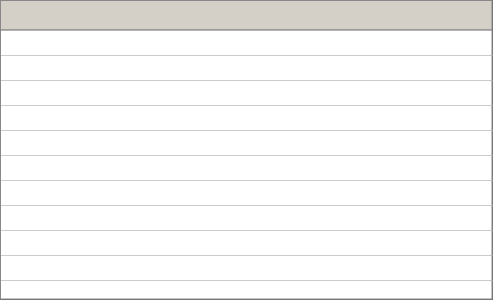
VISUALIZATION _VISU_SRS  // 493x300
VAR_IN_OUT
	mInst : FB_SRS;
END_VAR
    Table (0,0 493x300), data array: mInst.sSrsList
        p3854506369: mInst.sSrsList[INDEX].bImplemented
        p1892666644: mInst.sSrsList[INDEX].sKey
        p338671338: mInst.sSrsList[INDEX].sDescription
        p2170511999: mInst.sSrsList[INDEX].sLink
        p2232123230: Impl.
END_VISUALIZATION

(* stored: Version 1.1.0.1, ProductVersion 3.1.4024.11
   Visu _VISU_SRS: Id {f11480c5-cbf4-4c3a-af96-a666f49e69fd} *)
